// TIA Portal V19 export
TYPE "TMeasuringCtrl"
// stored: Access Published
   STRUCT
      Rst : Bool;   // Reset alarms
      MeasureEnable : Bool;   // Enable measuring
      Mode : DInt;   // 0 - 4 = see MC Measuring input mode; 10 = Capture Next Edge
   END_STRUCT;
END_TYPE
